TEXTLIST EL2809_M_4
  1 = 'Pump C1' | chinese: '供墨泵C1' | Chinese: '供墨泵C1'
  2 = 'Pump C2' | chinese: '供墨泵C2' | Chinese: '供墨泵C2'
  3 = 'Pump Y1' | chinese: '供墨泵Y1' | Chinese: '供墨泵Y1'
  4 = 'Pump Y2' | chinese: '供墨泵Y2' | Chinese: '供墨泵Y2'
  5 = 'Pump M1' | chinese: '供墨泵M1' | Chinese: '供墨泵M1'
  6 = 'Pump M2' | chinese: '供墨泵M2' | Chinese: '供墨泵M2'
  7 = 'Pump K1' | chinese: '供墨泵K1' | Chinese: '供墨泵K1'
  8 = 'Pump K2' | chinese: '供墨泵K2' | Chinese: '供墨泵K2'
  9 = 'Pump LC1' | chinese: '供墨泵LC1' | Chinese: '供墨泵LC1'
  10 = 'Pump LC2' | chinese: '供墨泵LC2' | Chinese: '供墨泵LC2'
  11 = 'Pump LM1' | chinese: '供墨泵LM1' | Chinese: '供墨泵LM1'
  12 = 'Pump LM2' | chinese: '供墨泵LM2' | Chinese: '供墨泵LM2'
  13 = 'Pump P1' | chinese: '图层泵 P1' | Chinese: '供墨泵 W1'
  14 = 'Pump P2' | chinese: '图层泵 P2' | Chinese: '供墨泵 W2'
  15 = 'Pump W1' | chinese: '供墨泵W1' | Chinese: '清洗液泵1'
  16 = 'Pump W2' | chinese: '供墨泵W2' | Chinese: '清洗液泵2'
   = ''
END_TEXTLIST

(* stored: Version 1.1.0.1, ProductVersion 3.1.4024.11
   TextList EL2809_M_4: Id {4c0abf45-40c5-4928-98c9-95a6a888e007} *)
